(* CoDeSys 2.3.9.31 project: AxisTest20170221.pro *)
(* Libraries: TcBase.lib 14.5.09 11:14:08, TcSystem.lib 27.2.12 14:08:36, TcBaseMath.lib 27.7.04 11:07:56, TcMath.lib 23.9.04 14:15:30, TcMC2.lib 23.8.12 10:01:14, STANDARD.LIB 5.6.98 11:03:02 *)

(* Task configuration *)
TASK Standard (PRIORITY := 0, INTERVAL := T#10ms);
	MAIN
END_TASK

(* Global variable list: Global_Variables *)
VAR_GLOBAL
	Axis1	:	Axis_Ref;
END_VAR

(* Global variable list: TwinCAT_Configuration *)
(* Generated automatically by TwinCAT - (read only) *)
VAR_CONFIG
	MAIN.HomeSign1 AT %IX128.0 : BOOL;	(*  ~ {LinkedWith:TIID^Device 2 (EtherCAT)^Term 1 (EK1100)^Term 2 (EL1889)^Channel 1^Input} *)
	.Axis1.PlcToNc AT %QB0 : PLCTONC_AXIS_REF;	(*  ~ {LinkedWith:TINC^NC-Task 1 SAF^Axes^Axis 1^Inputs^Axis 1_FromPlc} *)
	.Axis1.NcToPlc AT %IB0 : NCTOPLC_AXIS_REF;	(*  ~ {LinkedWith:TINC^NC-Task 1 SAF^Axes^Axis 1^Outputs^Axis 1_ToPlc} *)
END_VAR

(* POU MAIN, LD *)
PROGRAM MAIN

VAR
	HomeSign1 AT %I*	:	BOOL;
	M0: BOOL;
	HomeAction1: MC_Home;
	M1: BOOL;
	M2: BOOL;
	M3: BOOL;
	PowerAction1: MC_Power;
	M4: BOOL;
	ResetAction1: MC_Reset;
	M5: BOOL;
	HomeRDY: BOOL;
	R_TRIG1: R_TRIG;
	PowerOn: BOOL;
	M6: BOOL;
	MoveAbs1: MC_MoveAbsolute;
	P1: LREAL;
	M7: BOOL;
	V1: LREAL;
	M8: BOOL;
	M9: BOOL;
	M10: BOOL;
	TON1: TON;
	M12: BOOL;
	M13: BOOL;
	M14: BOOL;
	TON2: TON;
	M15: BOOL;
	ActPos1: LREAL;
	Error1: BOOL;
	ErrorID1: UDINT;
	M16: BOOL;
	MC_Jog1: MC_Jog;
	M17: BOOL;
	M19: BOOL;
	Mode1: UINT;
	M20: BOOL;
	M21: BOOL;
END_VAR
VAR (* helpers for the ST form of the networks *)
	_p1 : BOOL;
	_p2 : BOOL;
	_p3 : BOOL;
	_p4 : BOOL;
	_p5 : BOOL;
	_p6 : BOOL;
END_VAR
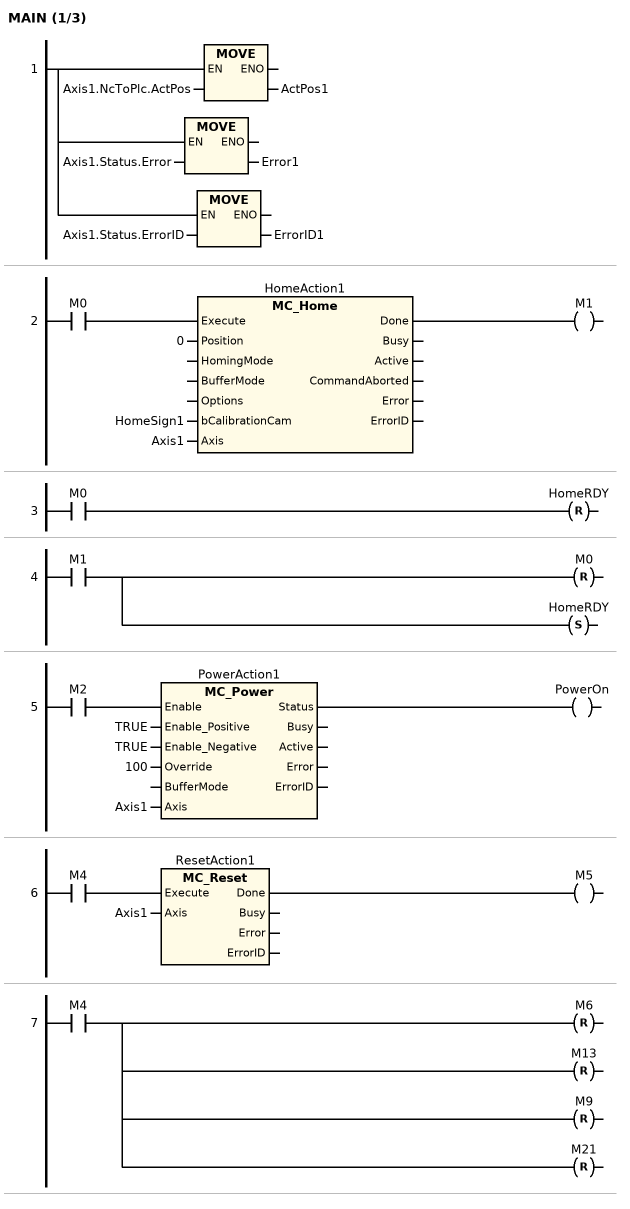
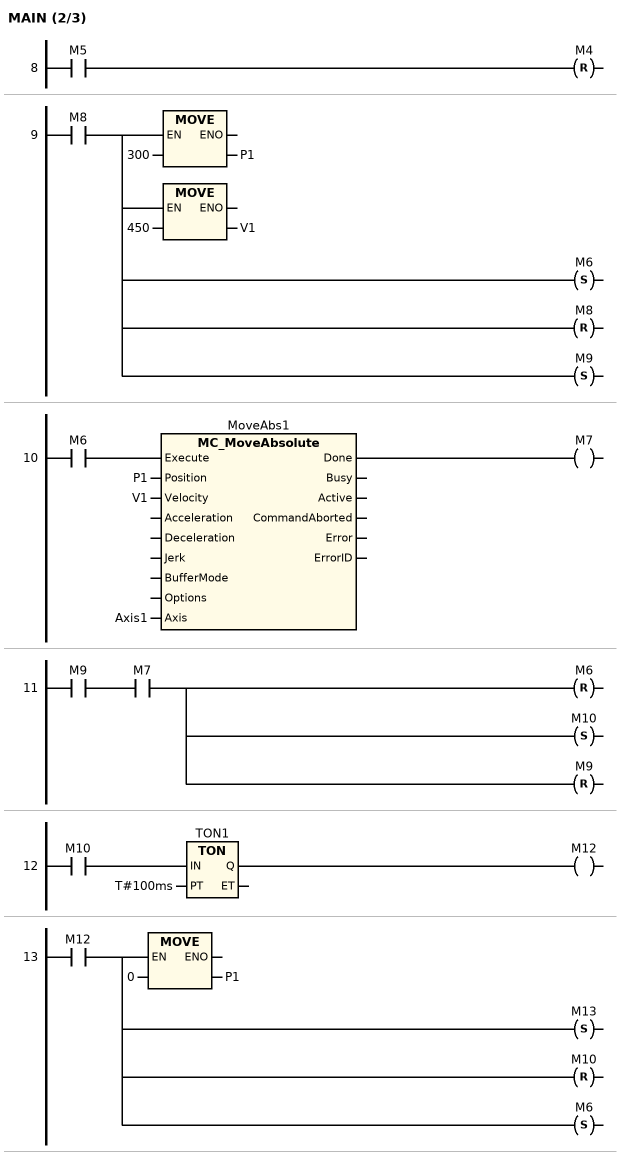
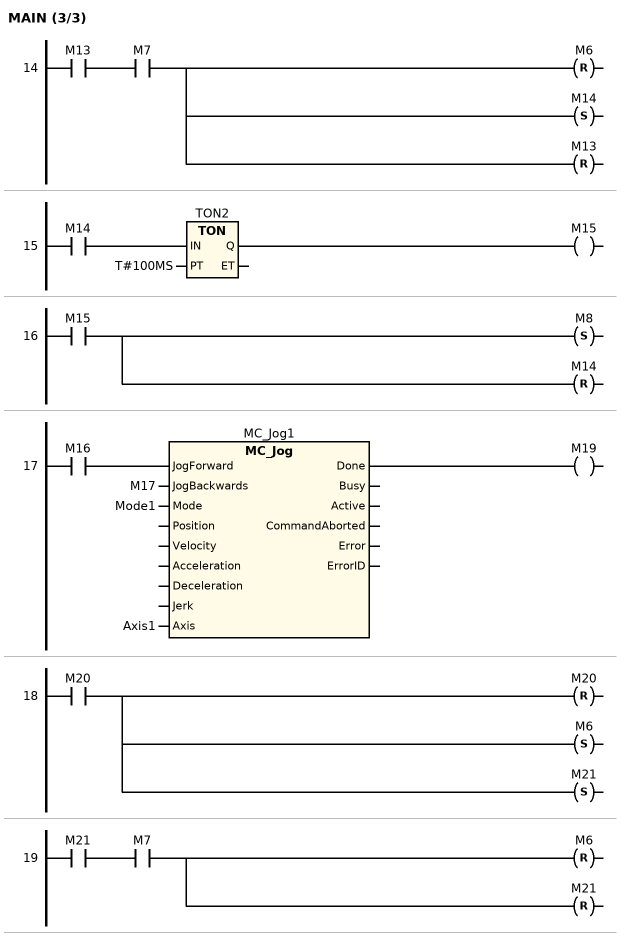
_LD_ (* Ladder Diagram *)
NETWORK 1
	*
		EN --- MOVE(Axis1.NcToPlc.ActPos) => ActPos1
		EN --- MOVE(Axis1.Status.Error) => Error1
		EN --- MOVE(Axis1.Status.ErrorID) => ErrorID1
NETWORK 2
	[M0] - HomeAction1:MC_Home(Execute: *, Position: 0, HomingMode: , BufferMode: , Options: , bCalibrationCam: HomeSign1, Axis: Axis1) --- (M1)
NETWORK 3
	[M0] --- (R HomeRDY)
NETWORK 4
	[M1] --- (R M0) (S HomeRDY)
NETWORK 5
	[M2] - PowerAction1:MC_Power(Enable: *, Enable_Positive: TRUE, Enable_Negative: TRUE, Override: 100, BufferMode: , Axis: Axis1) --- (PowerOn)
NETWORK 6
	[M4] - ResetAction1:MC_Reset(Execute: *, Axis: Axis1) --- (M5)
NETWORK 7
	[M4] --- (R M6) (R M13) (R M9) (R M21)
NETWORK 8
	[M5] --- (R M4)
NETWORK 9
	[M8] --- (S M6) (R M8) (S M9)
		EN --- MOVE(300) => P1
		EN --- MOVE(450) => V1
NETWORK 10
	[M6] - MoveAbs1:MC_MoveAbsolute(Execute: *, Position: P1, Velocity: V1, Acceleration: , Deceleration: , Jerk: , BufferMode: , Options: , Axis: Axis1) --- (M7)
NETWORK 11
	[M9] - [M7] --- (R M6) (S M10) (R M9)
NETWORK 12
	[M10] - TON1:TON(IN: *, PT: T#100ms) --- (M12)
NETWORK 13
	[M12] --- (S M13) (R M10) (S M6)
		EN --- MOVE(0) => P1
NETWORK 14
	[M13] - [M7] --- (R M6) (S M14) (R M13)
NETWORK 15
	[M14] - TON2:TON(IN: *, PT: T#100MS) --- (M15)
NETWORK 16
	[M15] --- (S M8) (R M14)
NETWORK 17
	[M16] - MC_Jog1:MC_Jog(JogForward: *, JogBackwards: M17, Mode: Mode1, Position: , Velocity: , Acceleration: , Deceleration: , Jerk: , Axis: Axis1) --- (M19)
NETWORK 18
	[M20] --- (R M20) (S M6) (S M21)
NETWORK 19
	[M21] - [M7] --- (R M6) (R M21)
_END_LD_
(* the same logic as Structured Text *)
(* Network 1 *)
ActPos1 := Axis1.NcToPlc.ActPos;
Error1 := Axis1.Status.Error;
ErrorID1 := Axis1.Status.ErrorID;
(* Network 2: see the listing above *)
(* Network 3 *)
IF M0 THEN HomeRDY := FALSE; END_IF;
(* Network 4 *)
IF M1 THEN M0 := FALSE; HomeRDY := TRUE; END_IF;
(* Network 5: see the listing above *)
(* Network 6 *)
ResetAction1(Execute := M4, Axis := Axis1);
M5 := ResetAction1.Done;
(* Network 7 *)
IF M4 THEN M6 := FALSE; M13 := FALSE; M9 := FALSE; M21 := FALSE; END_IF;
(* Network 8 *)
IF M5 THEN M4 := FALSE; END_IF;
(* Network 9 *)
_p1 := M8;
IF _p1 THEN
	P1 := 300;
	V1 := 450;
END_IF;
IF _p1 THEN M6 := TRUE; M8 := FALSE; M9 := TRUE; END_IF;
(* Network 10: see the listing above *)
(* Network 11 *)
_p2 := M9 AND M7;
IF _p2 THEN M6 := FALSE; M10 := TRUE; M9 := FALSE; END_IF;
(* Network 12 *)
TON1(IN := M10, PT := T#100ms);
M12 := TON1.Q;
(* Network 13 *)
_p3 := M12;
IF _p3 THEN
	P1 := 0;
END_IF;
IF _p3 THEN M13 := TRUE; M10 := FALSE; M6 := TRUE; END_IF;
(* Network 14 *)
_p4 := M13 AND M7;
IF _p4 THEN M6 := FALSE; M14 := TRUE; M13 := FALSE; END_IF;
(* Network 15 *)
TON2(IN := M14, PT := T#100MS);
M15 := TON2.Q;
(* Network 16 *)
IF M15 THEN M8 := TRUE; M14 := FALSE; END_IF;
(* Network 17: see the listing above *)
(* Network 18 *)
_p5 := M20;
IF _p5 THEN M20 := FALSE; M6 := TRUE; M21 := TRUE; END_IF;
(* Network 19 *)
_p6 := M21 AND M7;
IF _p6 THEN M6 := FALSE; M21 := FALSE; END_IF;
END_PROGRAM
